PROGRAM HoldingBit_DoorTransfer
VAR

	ARfbStnDoorCtrl		: ARRAY [1..iStnQty] OF fbSlidingDoorCtrl;
	ARfbStnDoorOpen		: ARRAY [1..iStnQty] OF CMP_OC_W1;
	ARfbStnDoorClose	: ARRAY [1..iStnQty] OF CMP_OC_W1;
	
	ARfbUldDoorCtrl		:  fbSlidingDoorCtrl;
	ARfbUldDoorOpen		:  CMP_OC_W1;
	ARfbUldDoorClose	:  CMP_OC_W1;
	
	ARfbUldConveyorCtrl		:  fbSlidingDoorCtrl;
	ARfbUldConveyorOpen		:  CMP_OC_W1;
	ARfbUldConveyorClose	:  CMP_OC_W1;
	
	

	LdDoorCtrl: fbSlidingDoorCtrl;
	LdDoorOpen: CMP_OC_W1;
	LdDoorClose: CMP_OC_W1;

	UldDoorCtrl: fbSlidingDoorCtrl;
	UldDoorOpen: CMP_OC_W1;
	UldDoorClose: CMP_OC_W1;

	bArm1TransferToStn1: BOOL;
	bArm1TransferToStn2: BOOL;
	bArm1TransferToStn3 : BOOL;
	bArm1TransferToStn4 : BOOL;
	bArm1TransferToStn5 : BOOL;
	bArm1TransferToStn6: BOOL;
	bArm1TransferToStn7: BOOL;
	bArm1TransferToStn8 : BOOL;
	bArm1TransferToStn9 : BOOL;
	bArm1TransferToStn10 : BOOL;
	bArm1TransferToStn11 : BOOL;
	bArm1TransferToStn12 : BOOL;
	bArm1TransferToUld1: BOOL;

	bArm2TransferToStn8 : BOOL;
	bArm2TransferToStn9 : BOOL;
	bArm2TransferToStn10 : BOOL;
	bArm2TransferToStn11 : BOOL;

	bArmPnpStep6: BOOL;

	TON1: TON;
	TON2: TON;
	TON3: TON;
	TON4: TON;
	TON5: TON;
	TON6: TON;
	TON7: TON;
	TON8: TON;
	TON9: TON;
	TON10: TON;
	TON11: TON;
	TON12: TON;
	TON13: TON;
	TON14: TON;
	TON15: TON;
	TON16: TON;
	TON17: TON;
	TON18: TON;
	TON19: TON;
	TON20: TON;
	TON21: TON;
	TON22: TON;
	TON23: TON;
	TON24: TON;
	TON25: TON;
	TON26: TON;
	TON27: TON;
	TON28: TON;
	TON29: TON;
	TON30: TON;
	
END_VAR

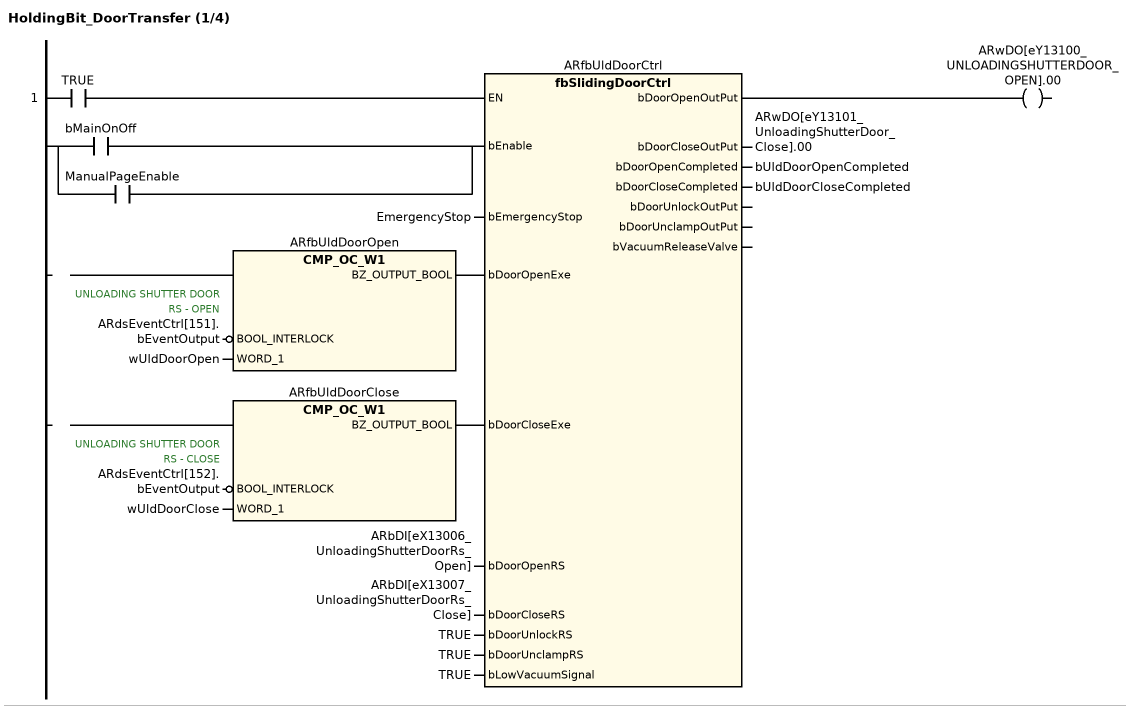
// NETWORK 1
//   ARdsEventCtrl[151].bEventOutput: UNLOADING SHUTTER DOOR RS - OPEN
//   ARdsEventCtrl[152].bEventOutput: UNLOADING SHUTTER DOOR RS - CLOSE
ARfbUldDoorOpen(BOOL_INTERLOCK := NOT ARdsEventCtrl[151].bEventOutput, WORD_1 := wUldDoorOpen); // CMP_OC_W1
ARfbUldDoorClose(BOOL_INTERLOCK := NOT ARdsEventCtrl[152].bEventOutput, WORD_1 := wUldDoorClose); // CMP_OC_W1
ARfbUldDoorCtrl(
    bEnable := bMainOnOff OR ManualPageEnable,
    bEmergencyStop := EmergencyStop,
    bDoorOpenExe := ARfbUldDoorOpen.BZ_OUTPUT_BOOL,
    bDoorCloseExe := ARfbUldDoorClose.BZ_OUTPUT_BOOL,
    bDoorOpenRS := ARbDI[eX13006_UnloadingShutterDoorRs_Open],
    bDoorCloseRS := ARbDI[eX13007_UnloadingShutterDoorRs_Close],
    bDoorUnlockRS := TRUE,
    bDoorUnclampRS := TRUE,
    bLowVacuumSignal := TRUE,
    bDoorCloseOutPut => ARwDO[eY13101_UnloadingShutterDoor_Close].00,
    bDoorOpenCompleted => bUldDoorOpenCompleted,
    bDoorCloseCompleted => bUldDoorCloseCompleted); // fbSlidingDoorCtrl
ARwDO[eY13100_UNLOADINGSHUTTERDOOR_OPEN].00 := ARfbUldDoorCtrl.bDoorOpenOutPut;

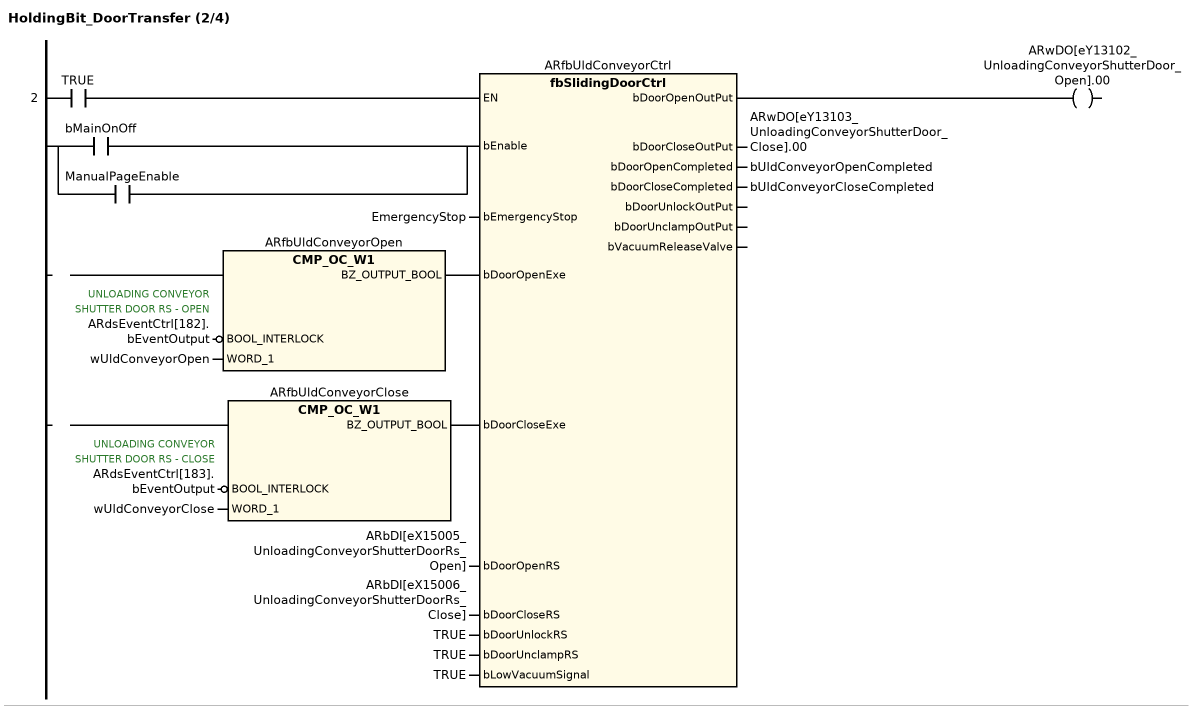
// NETWORK 2
//   ARdsEventCtrl[182].bEventOutput: UNLOADING CONVEYOR SHUTTER DOOR RS - OPEN
//   ARdsEventCtrl[183].bEventOutput: UNLOADING CONVEYOR SHUTTER DOOR RS - CLOSE
ARfbUldConveyorOpen(BOOL_INTERLOCK := NOT ARdsEventCtrl[182].bEventOutput, WORD_1 := wUldConveyorOpen); // CMP_OC_W1
ARfbUldConveyorClose(BOOL_INTERLOCK := NOT ARdsEventCtrl[183].bEventOutput, WORD_1 := wUldConveyorClose); // CMP_OC_W1
ARfbUldConveyorCtrl(
    bEnable := bMainOnOff OR ManualPageEnable,
    bEmergencyStop := EmergencyStop,
    bDoorOpenExe := ARfbUldConveyorOpen.BZ_OUTPUT_BOOL,
    bDoorCloseExe := ARfbUldConveyorClose.BZ_OUTPUT_BOOL,
    bDoorOpenRS := ARbDI[eX15005_UnloadingConveyorShutterDoorRs_Open],
    bDoorCloseRS := ARbDI[eX15006_UnloadingConveyorShutterDoorRs_Close],
    bDoorUnlockRS := TRUE,
    bDoorUnclampRS := TRUE,
    bLowVacuumSignal := TRUE,
    bDoorCloseOutPut => ARwDO[eY13103_UnloadingConveyorShutterDoor_Close].00,
    bDoorOpenCompleted => bUldConveyorOpenCompleted,
    bDoorCloseCompleted => bUldConveyorCloseCompleted); // fbSlidingDoorCtrl
ARwDO[eY13102_UnloadingConveyorShutterDoor_Open].00 := ARfbUldConveyorCtrl.bDoorOpenOutPut;

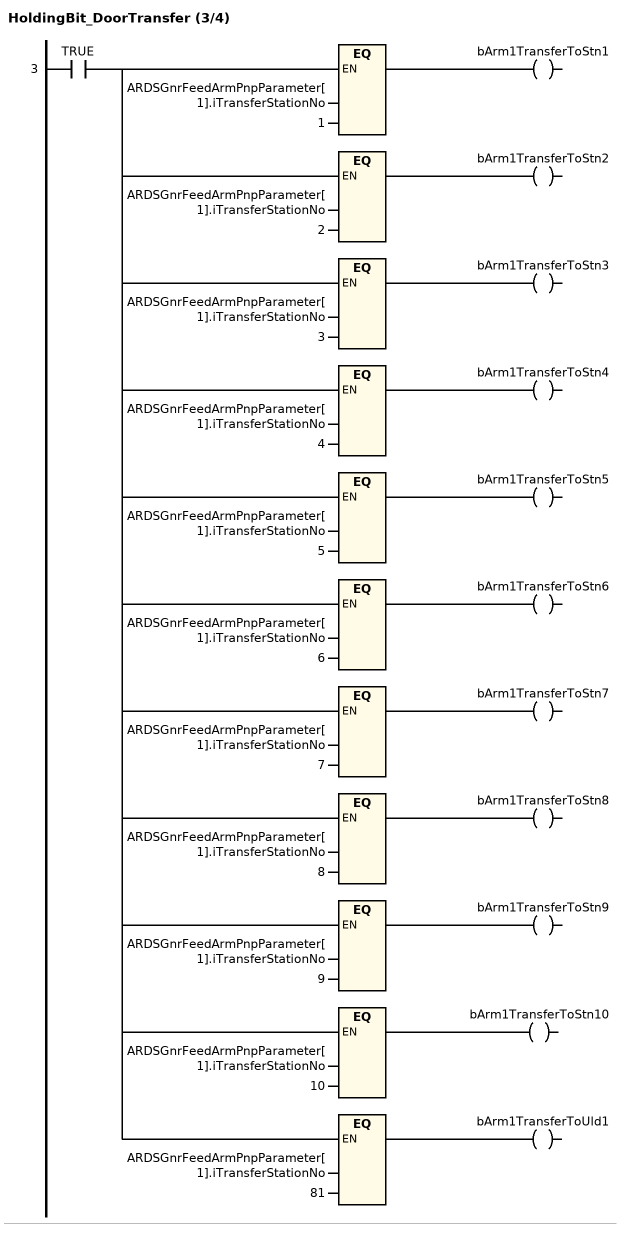
// NETWORK 3
bArm1TransferToStn1 := ARDSGnrFeedArmPnpParameter[1].iTransferStationNo = 1;
bArm1TransferToStn2 := ARDSGnrFeedArmPnpParameter[1].iTransferStationNo = 2;
bArm1TransferToStn3 := ARDSGnrFeedArmPnpParameter[1].iTransferStationNo = 3;
bArm1TransferToStn4 := ARDSGnrFeedArmPnpParameter[1].iTransferStationNo = 4;
bArm1TransferToStn5 := ARDSGnrFeedArmPnpParameter[1].iTransferStationNo = 5;
bArm1TransferToStn6 := ARDSGnrFeedArmPnpParameter[1].iTransferStationNo = 6;
bArm1TransferToStn7 := ARDSGnrFeedArmPnpParameter[1].iTransferStationNo = 7;
bArm1TransferToStn8 := ARDSGnrFeedArmPnpParameter[1].iTransferStationNo = 8;
bArm1TransferToStn9 := ARDSGnrFeedArmPnpParameter[1].iTransferStationNo = 9;
bArm1TransferToStn10 := ARDSGnrFeedArmPnpParameter[1].iTransferStationNo = 10;
bArm1TransferToUld1 := ARDSGnrFeedArmPnpParameter[1].iTransferStationNo = 81;

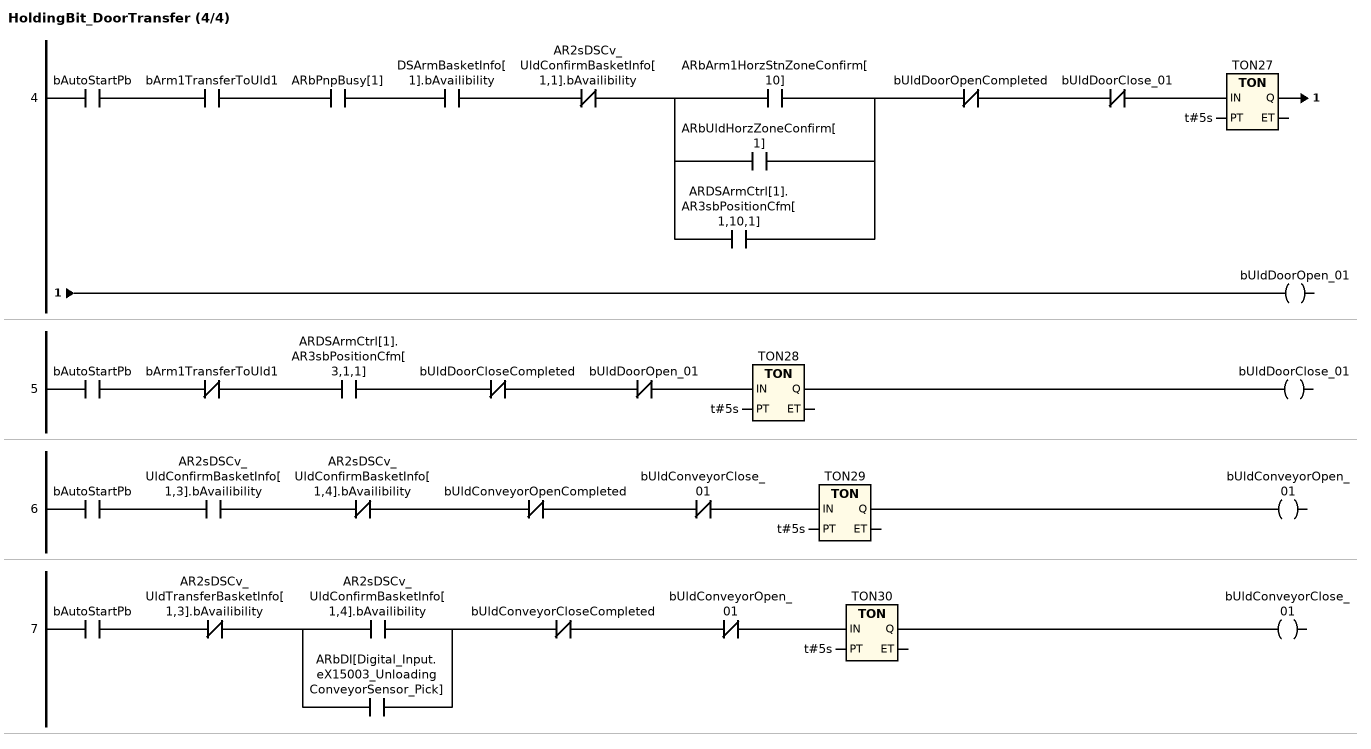
// NETWORK 4
TON27(IN := bAutoStartPb AND bArm1TransferToUld1 AND ARbPnpBusy[1] AND DSArmBasketInfo[1].bAvailibility AND NOT AR2sDSCv_UldConfirmBasketInfo[1,1].bAvailibility AND (ARbArm1HorzStnZoneConfirm[10] OR ARbUldHorzZoneConfirm[1] OR ARDSArmCtrl[1].AR3sbPositionCfm[1,10,1]) AND NOT bUldDoorOpenCompleted AND NOT bUldDoorClose_01, PT := t#5s); // TON
bUldDoorOpen_01 := TON27.Q;

// NETWORK 5
TON28(IN := bAutoStartPb AND NOT bArm1TransferToUld1 AND ARDSArmCtrl[1].AR3sbPositionCfm[3,1,1] AND NOT bUldDoorCloseCompleted AND NOT bUldDoorOpen_01, PT := t#5s); // TON
bUldDoorClose_01 := TON28.Q;

// NETWORK 6
TON29(IN := bAutoStartPb AND AR2sDSCv_UldConfirmBasketInfo[1,3].bAvailibility AND NOT AR2sDSCv_UldConfirmBasketInfo[1,4].bAvailibility AND NOT bUldConveyorOpenCompleted AND NOT bUldConveyorClose_01, PT := t#5s); // TON
bUldConveyorOpen_01 := TON29.Q;

// NETWORK 7
TON30(IN := bAutoStartPb AND NOT AR2sDSCv_UldTransferBasketInfo[1,3].bAvailibility AND (AR2sDSCv_UldConfirmBasketInfo[1,4].bAvailibility OR ARbDI[Digital_Input.eX15003_UnloadingConveyorSensor_Pick]) AND NOT bUldConveyorCloseCompleted AND NOT bUldConveyorOpen_01, PT := t#5s); // TON
bUldConveyorClose_01 := TON30.Q;

END_PROGRAM

(* stored: Version 1.1.0.1, ProductVersion 3.1.4024.12
   POU HoldingBit_DoorTransfer: Id {e1261944-0a43-42ec-b5af-7a08d6db97ad}, SpecialFunc None *)
